PROGRAM ValveManualControl
VAR
END_VAR

// written 18.08.2023 by Daniel Kelly

// Program provides manual control for the valves
// Valve1Open opens the top valve
// Valve1Close closes the top valve
// Valve2Open opens the bottom valve
// Valve2Close closes the bottom valve

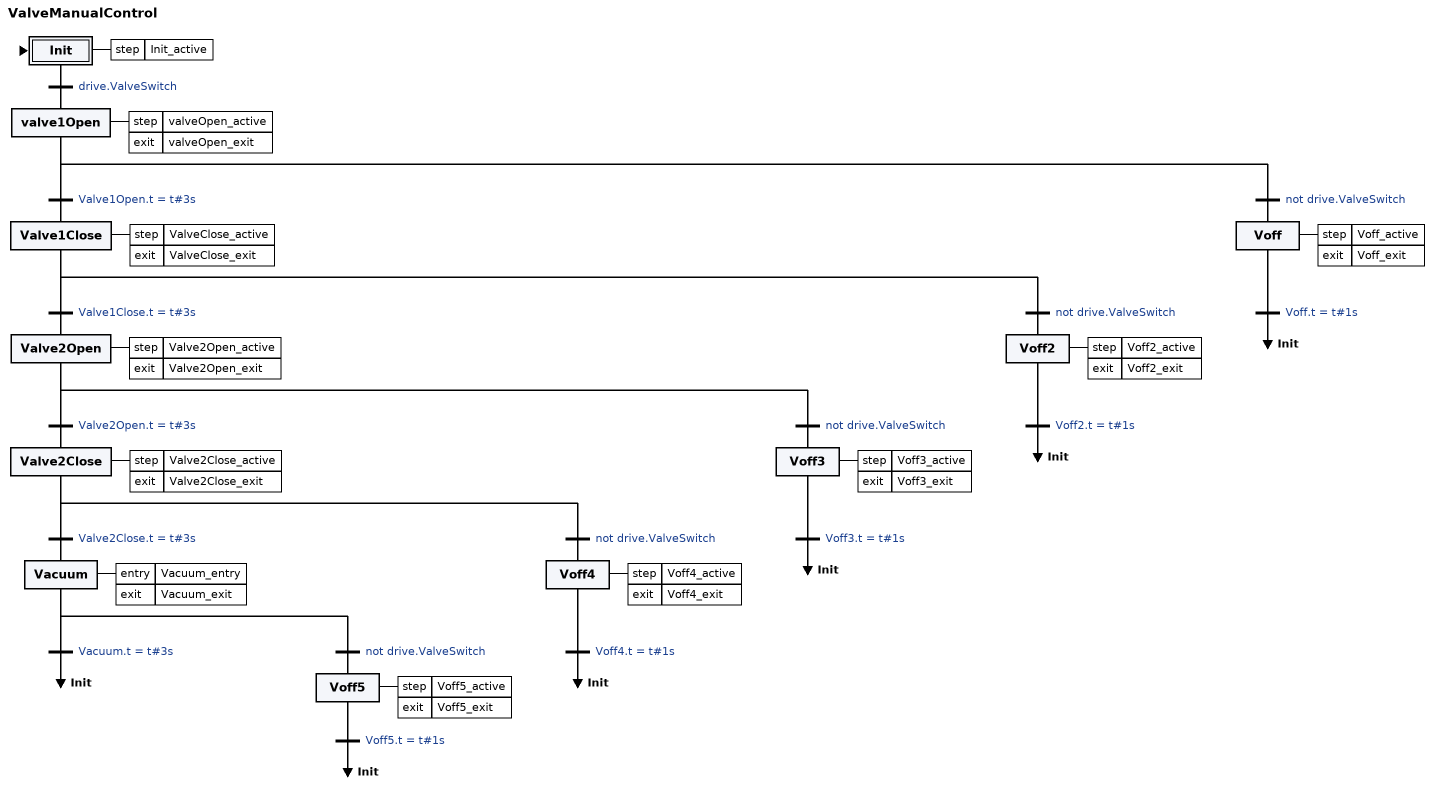
INITIAL_STEP Init:
    Init_active(N);  // step action
END_STEP
TRANSITION FROM Init TO valve1Open
    := drive.ValveSwitch;
END_TRANSITION
STEP valve1Open:
    valveOpen_active(N);  // step action
    valveOpen_exit(P0);  // exit action
END_STEP
TRANSITION FROM valve1Open TO Valve1Close
    := Valve1Open.t = t#3s;
END_TRANSITION
TRANSITION FROM valve1Open TO Voff
    := not drive.ValveSwitch;
END_TRANSITION
STEP Voff:
    Voff_active(N);  // step action
    Voff_exit(P0);  // exit action
END_STEP
TRANSITION FROM Voff TO Init
    := Voff.t = t#1s;
END_TRANSITION
STEP Valve1Close:
    ValveClose_active(N);  // step action
    ValveClose_exit(P0);  // exit action
END_STEP
TRANSITION FROM Valve1Close TO Valve2Open
    := Valve1Close.t = t#3s;
END_TRANSITION
TRANSITION FROM Valve1Close TO Voff2
    := not drive.ValveSwitch;
END_TRANSITION
STEP Voff2:
    Voff2_active(N);  // step action
    Voff2_exit(P0);  // exit action
END_STEP
TRANSITION FROM Voff2 TO Init
    := Voff2.t = t#1s;
END_TRANSITION
STEP Valve2Open:
    Valve2Open_active(N);  // step action
    Valve2Open_exit(P0);  // exit action
END_STEP
TRANSITION FROM Valve2Open TO Valve2Close
    := Valve2Open.t = t#3s;
END_TRANSITION
TRANSITION FROM Valve2Open TO Voff3
    := not drive.ValveSwitch;
END_TRANSITION
STEP Voff3:
    Voff3_active(N);  // step action
    Voff3_exit(P0);  // exit action
END_STEP
TRANSITION FROM Voff3 TO Init
    := Voff3.t = t#1s;
END_TRANSITION
STEP Valve2Close:
    Valve2Close_active(N);  // step action
    Valve2Close_exit(P0);  // exit action
END_STEP
TRANSITION FROM Valve2Close TO Vacuum
    := Valve2Close.t = t#3s;
END_TRANSITION
TRANSITION FROM Valve2Close TO Voff4
    := not drive.ValveSwitch;
END_TRANSITION
STEP Voff4:
    Voff4_active(N);  // step action
    Voff4_exit(P0);  // exit action
END_STEP
TRANSITION FROM Voff4 TO Init
    := Voff4.t = t#1s;
END_TRANSITION
STEP Vacuum:
    Vacuum_entry(P1);  // entry action
    Vacuum_exit(P0);  // exit action
END_STEP
TRANSITION FROM Vacuum TO Init
    := Vacuum.t = t#3s;
END_TRANSITION
TRANSITION FROM Vacuum TO Voff5
    := not drive.ValveSwitch;
END_TRANSITION
STEP Voff5:
    Voff5_active(N);  // step action
    Voff5_exit(P0);  // exit action
END_STEP
TRANSITION FROM Voff5 TO Init
    := Voff5.t = t#1s;
END_TRANSITION

ACTION Init_active:
//drive.LeftSolenoid := FALSE;
//drive.LeftSolenoid2 := FALSE;
//drive.RightSolenoid := FALSE;
//drive.RightSolenoid2 := FALSE;
END_ACTION

ACTION Vacuum_entry:
drive.bVacuum := TRUE;
END_ACTION

ACTION Vacuum_exit:
drive.bVacuum := FALSE;
END_ACTION

ACTION Valve2Close_active:
drive.CloseBottomValve := TRUE;
END_ACTION

ACTION Valve2Close_exit:
drive.CloseBottomValve := FALSE;
drive.bValveLamp := FALSE;
END_ACTION

ACTION Valve2Open_active:
drive.OpenBottomValve := TRUE;
END_ACTION

ACTION Valve2Open_exit:
drive.OpenBottomValve := FALSE;
END_ACTION

ACTION ValveClose_active:
drive.OpenTopValve := FALSE;
drive.CloseTopValve := TRUE;
END_ACTION

ACTION ValveClose_exit:
drive.CloseTopValve := FALSE;
END_ACTION

ACTION valveOpen_active:
drive.OpenTopValve := TRUE;
END_ACTION

ACTION valveOpen_exit:
drive.OpenTopValve := FALSE;
END_ACTION

ACTION Voff_active:
drive.OpenTopValve := FALSE;
drive.CloseTopValve := TRUE;
drive.OpenBottomValve := FALSE;
drive.CloseBottomValve := TRUE;
END_ACTION

ACTION Voff_exit:
drive.CloseBottomValve := FALSE;
drive.CloseTopValve := FALSE;
END_ACTION

ACTION Voff2_active:
drive.OpenTopValve := FALSE;
drive.CloseTopValve := TRUE;
drive.OpenBottomValve := FALSE;
drive.CloseBottomValve := TRUE;
END_ACTION

ACTION Voff2_exit:
drive.CloseBottomValve := FALSE;
drive.CloseTopValve := FALSE;
END_ACTION

ACTION Voff3_active:
drive.OpenTopValve := FALSE;
drive.CloseTopValve := TRUE;
drive.OpenBottomValve := FALSE;
drive.CloseBottomValve := TRUE;
END_ACTION

ACTION Voff3_exit:
drive.CloseBottomValve := FALSE;
drive.CloseTopValve := FALSE;
END_ACTION

ACTION Voff4_active:
drive.OpenTopValve := FALSE;
drive.CloseTopValve := TRUE;
drive.OpenBottomValve := FALSE;
drive.CloseBottomValve := TRUE;
END_ACTION

ACTION Voff4_exit:
drive.CloseBottomValve := FALSE;
drive.CloseTopValve := FALSE;
END_ACTION

ACTION Voff5_active:
drive.OpenTopValve := FALSE;
drive.CloseTopValve := TRUE;
drive.OpenBottomValve := FALSE;
drive.CloseBottomValve := TRUE;
END_ACTION

ACTION Voff5_exit:
drive.CloseBottomValve := FALSE;
drive.CloseTopValve := FALSE;
END_ACTION

END_PROGRAM

(* stored: Version 1.1.0.1, ProductVersion 3.1.4024.12
   POU ValveManualControl: Id {29d9f5f1-1c65-46e5-b60b-48132d5449b9}, SpecialFunc None
   Action Init_active: Id {e02b50d0-5f6f-4c4f-9a19-2b191247fea3}
   Action Vacuum_entry: Id {2ddee134-83d3-4ab2-b114-972cc7c5d5e3}
   Action Vacuum_exit: Id {acd44106-dfcc-4016-9c93-3fee8381d039}
   Action Valve2Close_active: Id {becb321d-591a-4beb-8f22-18e17566e3e5}
   Action Valve2Close_exit: Id {59de9fb0-883c-42ca-a489-5de01c403be8}
   Action Valve2Open_active: Id {0809960d-a722-462a-baa2-c5f2d1a68e1f}
   Action Valve2Open_exit: Id {5de03ae4-6333-4f13-b9eb-d4a32ee2aeae}
   Action ValveClose_active: Id {71f44d90-6e07-4f39-be16-7251354993d0}
   Action ValveClose_exit: Id {f4eb7e9d-a44f-4bfa-a52d-7731e926d730}
   Action valveOpen_active: Id {b0178839-346d-4bd6-8d18-2b366b454e0a}
   Action valveOpen_exit: Id {80d5b9be-f02d-4bc2-82e2-f66799083643}
   Action Voff_active: Id {191369cc-aa4b-4125-b69c-3370165e6618}
   Action Voff_exit: Id {6fde1d79-0704-4c6b-a44c-1e00e852ba90}
   Action Voff2_active: Id {45548e3e-1563-4a68-9e0d-3b2fd3f16814}
   Action Voff2_exit: Id {ea6022a2-e21b-44a7-927a-cf0d940a091c}
   Action Voff3_active: Id {03c36bca-79bd-4409-8133-e06284f41c85}
   Action Voff3_exit: Id {fa31cfba-e8ef-4921-8f19-ac43ad3db169}
   Action Voff4_active: Id {08b7d4c6-3f89-4cb5-a672-4c564cf131e2}
   Action Voff4_exit: Id {6ad247c4-aac2-429c-9f70-ac7c40a37725}
   Action Voff5_active: Id {c9d33037-a274-42f4-ab33-b1e7234ab1b4}
   Action Voff5_exit: Id {ee969f76-44b8-4a84-ad43-3a83db0c17c3} *)
